// TIA Portal V19 export
FUNCTION_BLOCK "A0302_Rulliera_FB"   // FB64, LAD
// stored: MemoryReserve 100, SetENOAutomatically false
   VAR_INPUT
      AreaInterface : "AreaInterface";
      ZSI : "udt_ZoneSafetyInterface";
      DSI_Feed1 : "udt_DeviceSafetyInterface";
      DSI_Feed2 : "udt_DeviceSafetyInterface";
      Drive_Ax1 : "TAx_DriveInterface";
      Drive_Ax2 : "TAx_DriveInterface";
      DataIn : Struct
         Ax : "SpeedMachine_DataIn";
         Sens : Struct
            Coda { ExternalAccessible := 'False'; ExternalVisible := 'False'; ExternalWritable := 'False'} : Struct
               FTC_Rall : Bool;   // Sensori presenza materiale banco rallentamento ingresso
               FTC_Prox_Ing : Bool;   // Sensori presenza materiale banco limite ingresso
            END_STRUCT;
            Centro { ExternalAccessible := 'False'; ExternalVisible := 'False'; ExternalWritable := 'False'} : Struct
               FTC_Centrale : Bool;
            END_STRUCT;
         END_STRUCT;
      END_STRUCT;
      CIn { ExternalAccessible := 'False'; ExternalVisible := 'False'; ExternalWritable := 'False'} : Struct
         Manager : Struct
            Ax_1 : "SpeedMachine_CIn_Manager";
            Ax_2 : "SpeedMachine_CIn_Manager";
         END_STRUCT;
         SemiAut_Pb : Bool;
         P5 : Struct
            Sollevatori : "ValveMachine_COut";
            SpintoreLong : "ValveMachine_COut";
            Sens : Struct
               FTC_Ingombro_A0301 : Bool;   // 1614BF1 - I50.7
            END_STRUCT;
         END_STRUCT;
         Bordatrice : Struct
            StopBordatrice : Bool;   // Stop Bordatrice da controllo quota spazio rimanente su rulliera di coda
            ReadyForMove : Bool;   // Pronto al movimento
            StandbyBordatrice : Bool;
         END_STRUCT;
         Rulliera : Struct
            Centratori : "ValveMachine_COut";   // Chiusura Centratori
            Sollevamento : "ValveMachine_COut";   // Solleva centratori
            Coda : Struct
               Sens : Struct
                  FTC_Rall : Bool;   // Sensori presenza materiale banco rallentamento ingresso
                  FTC_Prox_Ing : Bool;   // Sensori presenza materiale banco limite ingresso
               END_STRUCT;
            END_STRUCT;
            Centro : Struct
               Sens : Struct
                  FTC_Centrale : Bool;   // 2010BF1 - I50.2
               END_STRUCT;
            END_STRUCT;
         END_STRUCT;
         CarroPareggCoda : Struct
            Ax : "Positioning_DOL_Machine_COut";
            Bloccaggio : "ValveMachine_COut";
            BattutaVerticale : "ValveMachine_COut";
            PareggiatoreLong : "ValveMachine_COut";
            Sens : Struct
               FTC_Ingombro_In : Bool;   // 2012BF1 - I50.0
               FTC_Ingombro_Out : Bool;   // 2012BF2 - I50.1
               PresenzaMat : Bool;   // FC presenza materiale agganciato lato paregg coda
               PosPareggLong : Struct
                  Value : LReal;
                  CheckMeasure : Bool;
                  Standstill : Bool;
               END_STRUCT;
            END_STRUCT;
         END_STRUCT;
         CarroPareggTesta : Struct
            Ax : "Positioning_DOL_Machine_COut";
            Bloccaggio : "ValveMachine_COut";
            Centraggio : "ValveMachine_COut";
            Sollevatore : "ValveMachine_COut";
            Sens : Struct
               FTC1_Rall : Bool;   // 2010BF2 - I50.3
               FTC2_Prox_Ls : Bool;   // 2010BF3 - I50.4
               PresenzaMat : Bool;   // FC presenza materiale agganciato lato paregg testa
            END_STRUCT;
         END_STRUCT;
         BTrk : Struct
            ZoneA0302Entry_Empty : Bool;
            ZoneA0302Exit_Empty : Bool;
         END_STRUCT;
      END_STRUCT;
      Config : Struct
         Ax : "SpeedMachine_Config";
      END_STRUCT;
      HWID_Ax_TEL1 : Array[1..2] of HW_SUBMODULE;
   END_VAR
   VAR_OUTPUT
      MachineInterface : "MachineInterface";
      COut : Struct
         Ax_1 : "SpeedMachine_COut";
         Ax_2 : "SpeedMachine_COut";
         Ax_VelOveride : Struct
            Enable : Bool;
            Value : Real;
         END_STRUCT;
      END_STRUCT;
   END_VAR
   VAR_IN_OUT
      Par : Struct
         Ax : "SpeedMachine_Par";
         Ax_Aut : "A0301_Mach_Speed_Par";
      END_STRUCT;
      IEC_SP : Struct
         FTC_CodaRall : Struct
            TON_PT : Time;
            TOF_PT : Time;
         END_STRUCT;
         FTC_CodaProx_Ing : Struct
            TON_PT : Time;
            TOF_PT : Time;
         END_STRUCT;
         FTC_Centro : Struct
            TON_PT : Time;
            TOF_PT : Time;
         END_STRUCT;
      END_STRUCT;
   END_VAR
   VAR
      Alarm : Struct
         Rulliera : Array[1..2] of "SpeedMachine_Alr";
      END_STRUCT;
      Warning : Struct
         Rulliera : Array[1..2] of "SpeedMachine_Wng";
         OP_REST_MissingCnd : Bool;   // Mancanza comando arresto
         OP_WORK_MissingCnd : Bool;   // Mancanza consenso lavoro
      END_STRUCT;
      HMI : Struct
         Selection : Struct   // 0=Disable / 1=Enable Pin
            Ax : Int;   // 0:Entrambe / 1:Rulliera Ax1 / 2:Rulliera Ax2
         END_STRUCT;
      END_STRUCT;
      Ax_1 : "SpeedMachine_FB";
      Ax_2 : "SpeedMachine_FB";
      ValueVelOvr { ExternalAccessible := 'False'; ExternalVisible := 'False'; ExternalWritable := 'False'} : Array[1..10] of Real;
      Sts : Struct
         OP_CanMoveFreely : Bool;
         OP_Bwd_Cnd : Bool;
         OP_Fwd_Cnd : Bool;
      END_STRUCT;
      Ctrl : Struct
         OP_Bwd_Man : Bool;
         OP_Fwd_Man : Bool;
         OP_Bwd_Aut : Bool;
         OP_Fwd_Aut : Bool;
         OP_Bwd_Run : Bool;
         OP_Fwd_Run : Bool;
      END_STRUCT;
      AUX : Struct
         OP_Bwd_PB : Bool;
         OP_Fwd_PB : Bool;
      END_STRUCT;
      TON_OP_REST_MissingCnd { S7_SetPoint := 'True'} : TON_TIME;
      TON_OP_WORK_MissingCnd { S7_SetPoint := 'True'} : TON_TIME;
      IEC_FTC_CodaRall : Struct
         TON_Delay : IEC_TIMER;
         TOF_Delay { S7_SetPoint := 'True'} : IEC_TIMER;
         FTC_On { S7_SetPoint := 'True'} : Bool;
      END_STRUCT;
      IEC_FTC_CodaProxIng : Struct
         TON_Delay : IEC_TIMER;
         TOF_Delay { S7_SetPoint := 'True'} : IEC_TIMER;
         FTC_On { S7_SetPoint := 'True'} : Bool;
      END_STRUCT;
      IEC_FTC_Centro : Struct
         TON_Delay : IEC_TIMER;
         TOF_Delay { S7_SetPoint := 'True'} : IEC_TIMER;
         FTC_On { S7_SetPoint := 'True'} : Bool;
      END_STRUCT;
   END_VAR
   VAR_TEMP
      PE : Struct
         OP_Bwd_PB : Bool;
         OP_Fwd_PB : Bool;
      END_STRUCT;
      VelOvr_Max : Real;   // Velocità max trovata
      i : Int;
      Check : Struct
         Cndz1_StartFwd : Bool;   // Check conditions to P4
         Cndz2_StartFwd : Bool;   // Check conditions to Allineatore laterale
      END_STRUCT;
   END_VAR
   VAR_TEMP   // added for the SCL form of the ladder/FBD networks
      _w1 : Bool;
      _w2 : Bool;
      _w3 : Bool;
   END_VAR
BEGIN

REGION Network 1 (SCL): == Riferimenti [Ax] - Speed Machine ==
   // ******************************************************************************************
   REGION // TRASFERIMENTO DELLE RAMPE

       // Rampe in Manuale
       IF #AreaInterface.Man AND NOT #CIn.SemiAut_Pb THEN
           #Ax_1.CIn.Manager.Vel := #Ax_2.CIn.Manager.Vel := #Par.Ax.Man.VelFwdHigh;
           #Ax_1.CIn.Manager.Acc :=  #Ax_2.CIn.Manager.Acc := #Par.Ax.Man.Acc;
           #Ax_1.CIn.Manager.Dec := #Ax_2.CIn.Manager.Dec := #Par.Ax.Man.Dec;
       END_IF;
   END_REGION

   // ******************************************************************************************
   REGION // CALCOLO DELLA VELOCITA' TRASFERITA DALL'IMPIANTO IN BASE ALLA LUNGHEZZA DEL PEZZO 

       // Inizializzo variabile di appoggio controllo overide massimo a un valore basso rispetto setpoint
       IF "Sys".AuxFirstPLCCycle THEN
           #VelOvr_Max := 100.0;
       END_IF;

       // Trasferisco le varibili su un array
       #ValueVelOvr[1] := "PPrf_MAIN".ON_WORK.A0301_A0302.Trasporto.VelOvr_PLen_UpTo_1000;
       #ValueVelOvr[2] := "PPrf_MAIN".ON_WORK.A0301_A0302.Trasporto.VelOvr_PLen_UpTo_1500;
       #ValueVelOvr[3] := "PPrf_MAIN".ON_WORK.A0301_A0302.Trasporto.VelOvr_PLen_UpTo_2000;
       #ValueVelOvr[4] := "PPrf_MAIN".ON_WORK.A0301_A0302.Trasporto.VelOvr_PLen_UpTo_2500;
       #ValueVelOvr[5] := "PPrf_MAIN".ON_WORK.A0301_A0302.Trasporto.VelOvr_PLen_UpTo_3000;
       #ValueVelOvr[6] := "PPrf_MAIN".ON_WORK.A0301_A0302.Trasporto.VelOvr_PLen_UpTo_3500;
       #ValueVelOvr[7] := "PPrf_MAIN".ON_WORK.A0301_A0302.Trasporto.VelOvr_PLen_UpTo_4000;
       #ValueVelOvr[8] := "PPrf_MAIN".ON_WORK.A0301_A0302.Trasporto.VelOvr_PLen_UpTo_4500;
       #ValueVelOvr[9] := "PPrf_MAIN".ON_WORK.A0301_A0302.Trasporto.VelOvr_PLen_UpTo_5000;
       #ValueVelOvr[10] := "PPrf_MAIN".ON_WORK.A0301_A0302.Trasporto.VelOvr_PLen_UpTo_5500;


       // Ciclo per verificare la variabile maggiore per prenderla in lavoro
       FOR #i := 1 TO 10 DO
           IF #ValueVelOvr[#i] >= #VelOvr_Max THEN
               #VelOvr_Max := #ValueVelOvr[#i];
           END_IF;
       END_FOR;
   END_REGION ;

   IF #VelOvr_Max = 0.0 THEN
       #VelOvr_Max := 100.0;
   END_IF;

   // ******************************************************************************************
   REGION // CALCOLO DELLA VELOCITA' E TRASFERIMENTO IN BASE ALLO STATO IMPIANTO

       #Ax_1.CIn.VelocityOverride.Enable := TRUE;
       #Ax_2.CIn.VelocityOverride.Enable := TRUE;

       IF #Ax_1.CIn.Manager.Control_ON THEN
           // CALCOLO VELOCITA' IN BASE ALL'OVERIDE
           #Ax_1.CIn.VelocityOverride.Value :=  #VelOvr_Max;
       ELSE
           #Ax_1.CIn.VelocityOverride.Value := 100.0;
           END_IF;

           IF #Ax_2.CIn.Manager.Control_ON THEN
               #Ax_2.CIn.VelocityOverride.Value := #VelOvr_Max;
           ELSE
               #Ax_2.CIn.VelocityOverride.Value := 100.0;
           END_IF;
       END_REGION ;
END_REGION

REGION Network 3: DataIn - FTC CodaRall
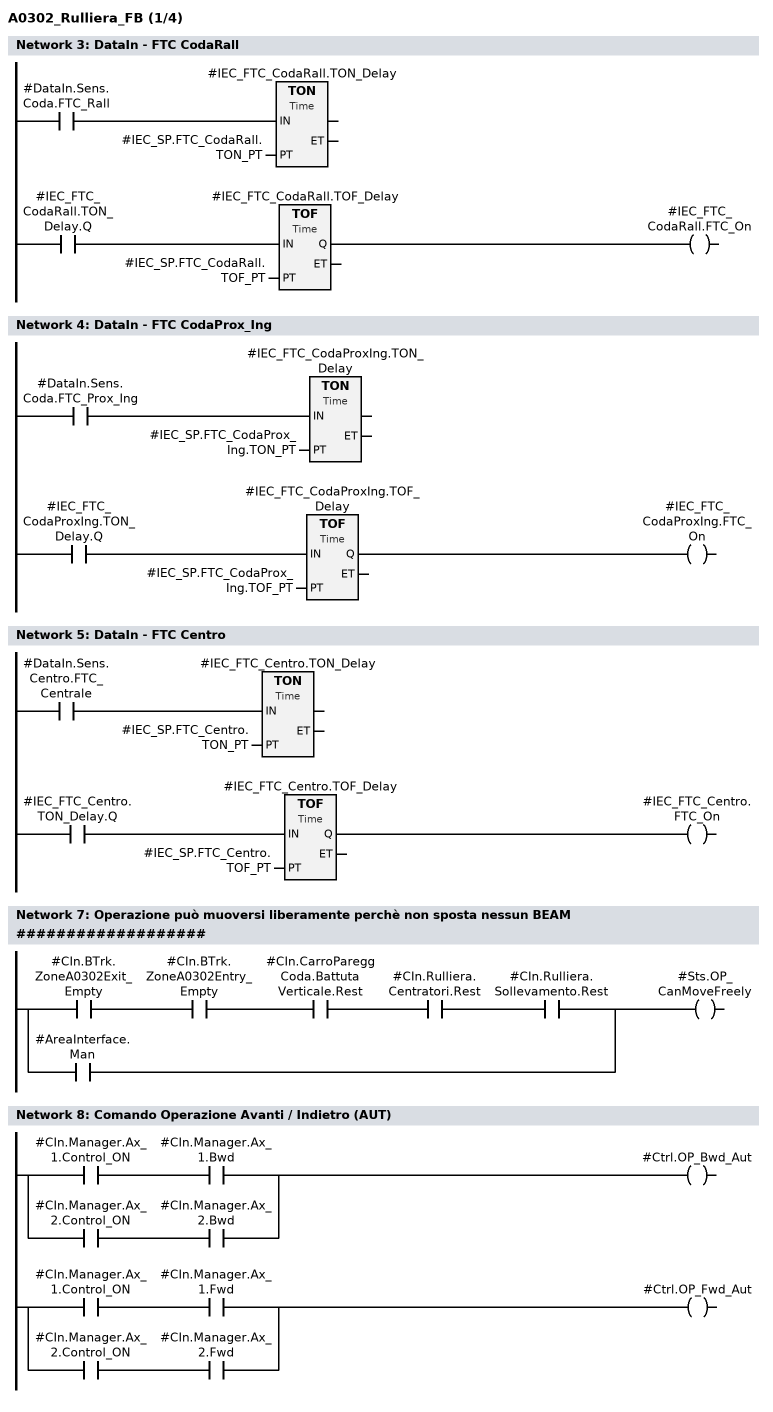
   RUNG wire#powerrail
      Contact( #DataIn.Sens.Coda.FTC_Rall )
      { S7_Templates := "time_type := Time" } #IEC_FTC_CodaRall.TON_Delay.TON(pt := #IEC_SP.FTC_CodaRall.TON_PT, et =>)
   END_RUNG
   RUNG wire#powerrail
      Contact( #IEC_FTC_CodaRall.TON_Delay.Q )
      { S7_Templates := "time_type := Time" } #IEC_FTC_CodaRall.TOF_Delay.TOF(pt := #IEC_SP.FTC_CodaRall.TOF_PT, et =>)
      Coil( #IEC_FTC_CodaRall.FTC_On )
   END_RUNG
   // the same network as SCL:
   #IEC_FTC_CodaRall.TON_Delay.TON(IN := #DataIn.Sens.Coda.FTC_Rall, PT := #IEC_SP.FTC_CodaRall.TON_PT);
   #IEC_FTC_CodaRall.TOF_Delay.TOF(IN := #IEC_FTC_CodaRall.TON_Delay.Q, PT := #IEC_SP.FTC_CodaRall.TOF_PT);
   #IEC_FTC_CodaRall.FTC_On := #IEC_FTC_CodaRall.TOF_Delay.Q;
END_REGION

REGION Network 4: DataIn - FTC CodaProx_Ing
   RUNG wire#powerrail
      Contact( #DataIn.Sens.Coda.FTC_Prox_Ing )
      { S7_Templates := "time_type := Time" } #IEC_FTC_CodaProxIng.TON_Delay.TON(pt := #IEC_SP.FTC_CodaProx_Ing.TON_PT, et =>)
   END_RUNG
   RUNG wire#powerrail
      Contact( #IEC_FTC_CodaProxIng.TON_Delay.Q )
      { S7_Templates := "time_type := Time" } #IEC_FTC_CodaProxIng.TOF_Delay.TOF(pt := #IEC_SP.FTC_CodaProx_Ing.TOF_PT, et =>)
      Coil( #IEC_FTC_CodaProxIng.FTC_On )
   END_RUNG
   // the same network as SCL:
   #IEC_FTC_CodaProxIng.TON_Delay.TON(IN := #DataIn.Sens.Coda.FTC_Prox_Ing,
                           PT := #IEC_SP.FTC_CodaProx_Ing.TON_PT);
   #IEC_FTC_CodaProxIng.TOF_Delay.TOF(IN := #IEC_FTC_CodaProxIng.TON_Delay.Q,
                           PT := #IEC_SP.FTC_CodaProx_Ing.TOF_PT);
   #IEC_FTC_CodaProxIng.FTC_On := #IEC_FTC_CodaProxIng.TOF_Delay.Q;
END_REGION

REGION Network 5: DataIn - FTC Centro
   RUNG wire#powerrail
      Contact( #DataIn.Sens.Centro.FTC_Centrale )
      { S7_Templates := "time_type := Time" } #IEC_FTC_Centro.TON_Delay.TON(pt := #IEC_SP.FTC_Centro.TON_PT, et =>)
   END_RUNG
   RUNG wire#powerrail
      Contact( #IEC_FTC_Centro.TON_Delay.Q )
      { S7_Templates := "time_type := Time" } #IEC_FTC_Centro.TOF_Delay.TOF(pt := #IEC_SP.FTC_Centro.TOF_PT, et =>)
      Coil( #IEC_FTC_Centro.FTC_On )
   END_RUNG
   // the same network as SCL:
   #IEC_FTC_Centro.TON_Delay.TON(IN := #DataIn.Sens.Centro.FTC_Centrale, PT := #IEC_SP.FTC_Centro.TON_PT);
   #IEC_FTC_Centro.TOF_Delay.TOF(IN := #IEC_FTC_Centro.TON_Delay.Q, PT := #IEC_SP.FTC_Centro.TOF_PT);
   #IEC_FTC_Centro.FTC_On := #IEC_FTC_Centro.TOF_Delay.Q;
END_REGION

REGION Network 7: Operazione può muoversi liberamente perchè non sposta nessun BEAM ###################
   RUNG wire#powerrail
      Contact( #CIn.BTrk.ZoneA0302Exit_Empty )
      Contact( #CIn.BTrk.ZoneA0302Entry_Empty )
      Contact( #CIn.CarroPareggCoda.BattutaVerticale.Rest )
      Contact( #CIn.Rulliera.Centratori.Rest )
      Contact( #CIn.Rulliera.Sollevamento.Rest )
      wire#w1
      Coil( #Sts.OP_CanMoveFreely )
   END_RUNG
   RUNG wire#powerrail
      Contact( #AreaInterface.Man )
   END_RUNG wire#w1
   // the same network as SCL:
   #Sts.OP_CanMoveFreely := (#CIn.BTrk.ZoneA0302Exit_Empty AND #CIn.BTrk.ZoneA0302Entry_Empty AND #CIn.CarroPareggCoda.BattutaVerticale.Rest AND #CIn.Rulliera.Centratori.Rest AND #CIn.Rulliera.Sollevamento.Rest) OR #AreaInterface.Man;
END_REGION

REGION Network 8: Comando Operazione Avanti / Indietro (AUT)
   RUNG wire#powerrail
      Contact( #CIn.Manager.Ax_1.Control_ON )
      Contact( #CIn.Manager.Ax_1.Bwd )
      wire#w1
      Coil( #Ctrl.OP_Bwd_Aut )
   END_RUNG
   RUNG wire#powerrail
      Contact( #CIn.Manager.Ax_2.Control_ON )
      Contact( #CIn.Manager.Ax_2.Bwd )
   END_RUNG wire#w1
   RUNG wire#powerrail
      Contact( #CIn.Manager.Ax_1.Control_ON )
      Contact( #CIn.Manager.Ax_1.Fwd )
      wire#w2
      Coil( #Ctrl.OP_Fwd_Aut )
   END_RUNG
   RUNG wire#powerrail
      Contact( #CIn.Manager.Ax_2.Control_ON )
      Contact( #CIn.Manager.Ax_2.Fwd )
   END_RUNG wire#w2
   // the same network as SCL:
   #Ctrl.OP_Bwd_Aut := (#CIn.Manager.Ax_1.Control_ON AND #CIn.Manager.Ax_1.Bwd) OR (#CIn.Manager.Ax_2.Control_ON AND #CIn.Manager.Ax_2.Bwd);
   #Ctrl.OP_Fwd_Aut := (#CIn.Manager.Ax_1.Control_ON AND #CIn.Manager.Ax_1.Fwd) OR (#CIn.Manager.Ax_2.Control_ON AND #CIn.Manager.Ax_2.Fwd);
END_REGION

REGION Network 9: Comando Operazione Lavoro / Riposo (MAN)
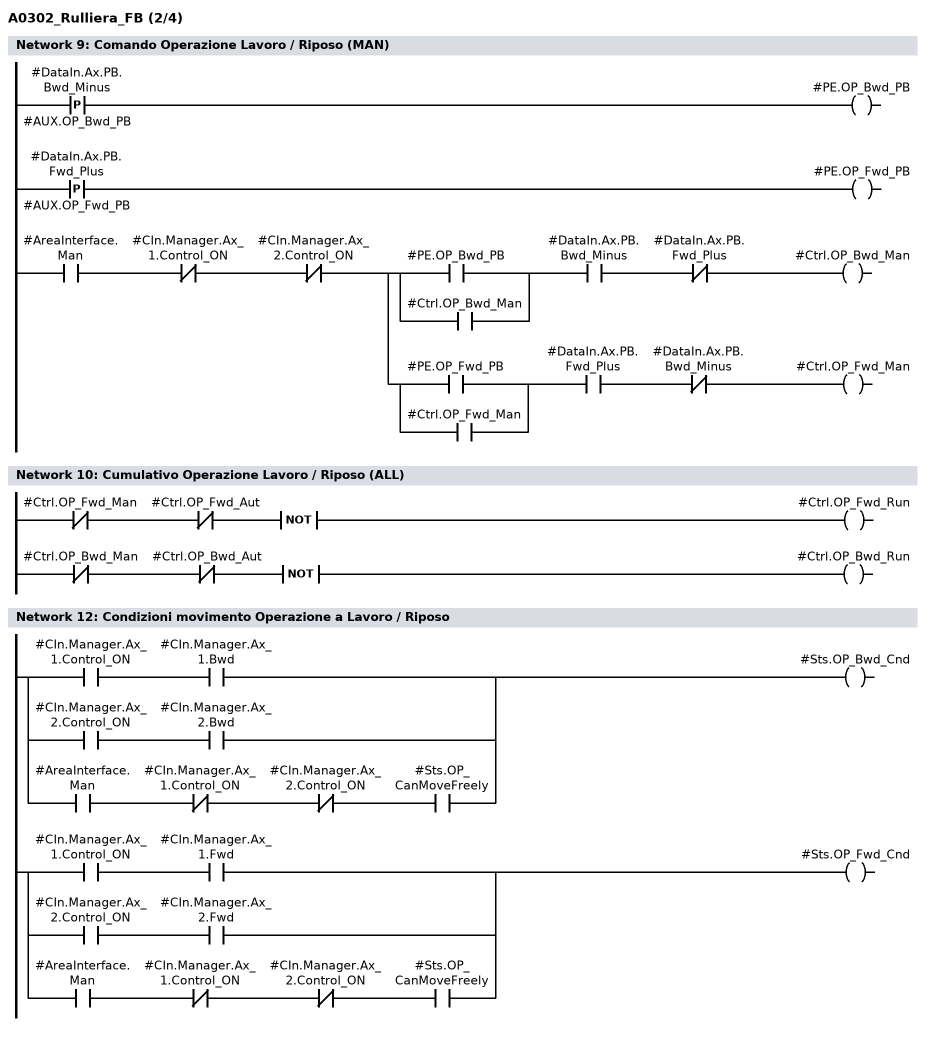
   RUNG wire#powerrail
      P_Contact(operand := #DataIn.Ax.PB.Bwd_Minus, bit := #AUX.OP_Bwd_PB)
      Coil( #PE.OP_Bwd_PB )
   END_RUNG
   RUNG wire#powerrail
      P_Contact(operand := #DataIn.Ax.PB.Fwd_Plus, bit := #AUX.OP_Fwd_PB)
      Coil( #PE.OP_Fwd_PB )
   END_RUNG
   RUNG wire#powerrail
      Contact( #AreaInterface.Man )
      I_Contact( #CIn.Manager.Ax_1.Control_ON )
      I_Contact( #CIn.Manager.Ax_2.Control_ON )
      wire#w1
      Contact( #PE.OP_Bwd_PB )
      wire#w2
      Contact( #DataIn.Ax.PB.Bwd_Minus )
      I_Contact( #DataIn.Ax.PB.Fwd_Plus )
      Coil( #Ctrl.OP_Bwd_Man )
   END_RUNG
   RUNG wire#w1
      Contact( #Ctrl.OP_Bwd_Man )
   END_RUNG wire#w2
   RUNG wire#w1
      Contact( #PE.OP_Fwd_PB )
      wire#w3
      Contact( #DataIn.Ax.PB.Fwd_Plus )
      I_Contact( #DataIn.Ax.PB.Bwd_Minus )
      Coil( #Ctrl.OP_Fwd_Man )
   END_RUNG
   RUNG wire#w1
      Contact( #Ctrl.OP_Fwd_Man )
   END_RUNG wire#w3
   // the same network as SCL:
   #_w1 := #DataIn.Ax.PB.Bwd_Minus AND NOT #AUX.OP_Bwd_PB;   // rising edge of #DataIn.Ax.PB.Bwd_Minus
   #AUX.OP_Bwd_PB := #DataIn.Ax.PB.Bwd_Minus;
   #PE.OP_Bwd_PB := #_w1;
   #_w2 := #DataIn.Ax.PB.Fwd_Plus AND NOT #AUX.OP_Fwd_PB;   // rising edge of #DataIn.Ax.PB.Fwd_Plus
   #AUX.OP_Fwd_PB := #DataIn.Ax.PB.Fwd_Plus;
   #PE.OP_Fwd_PB := #_w2;
   #_w3 := #AreaInterface.Man AND NOT #CIn.Manager.Ax_1.Control_ON AND NOT #CIn.Manager.Ax_2.Control_ON;
   #Ctrl.OP_Bwd_Man := #_w3 AND (#PE.OP_Bwd_PB OR #Ctrl.OP_Bwd_Man) AND #DataIn.Ax.PB.Bwd_Minus AND NOT #DataIn.Ax.PB.Fwd_Plus;
   #Ctrl.OP_Fwd_Man := #_w3 AND (#PE.OP_Fwd_PB OR #Ctrl.OP_Fwd_Man) AND #DataIn.Ax.PB.Fwd_Plus AND NOT #DataIn.Ax.PB.Bwd_Minus;
END_REGION

REGION Network 10: Cumulativo Operazione Lavoro / Riposo (ALL)
   RUNG wire#powerrail
      I_Contact( #Ctrl.OP_Fwd_Man )
      I_Contact( #Ctrl.OP_Fwd_Aut )
      Not()
      Coil( #Ctrl.OP_Fwd_Run )
   END_RUNG
   RUNG wire#powerrail
      I_Contact( #Ctrl.OP_Bwd_Man )
      I_Contact( #Ctrl.OP_Bwd_Aut )
      Not()
      Coil( #Ctrl.OP_Bwd_Run )
   END_RUNG
   // the same network as SCL:
   #Ctrl.OP_Fwd_Run := NOT (NOT #Ctrl.OP_Fwd_Man AND NOT #Ctrl.OP_Fwd_Aut);
   #Ctrl.OP_Bwd_Run := NOT (NOT #Ctrl.OP_Bwd_Man AND NOT #Ctrl.OP_Bwd_Aut);
END_REGION

REGION Network 11: <+>
END_REGION

REGION Network 12: Condizioni movimento Operazione a Lavoro / Riposo
   RUNG wire#powerrail
      Contact( #CIn.Manager.Ax_1.Control_ON )
      Contact( #CIn.Manager.Ax_1.Bwd )
      wire#w1
      Coil( #Sts.OP_Bwd_Cnd )
   END_RUNG
   RUNG wire#powerrail
      Contact( #CIn.Manager.Ax_2.Control_ON )
      Contact( #CIn.Manager.Ax_2.Bwd )
   END_RUNG wire#w1
   RUNG wire#powerrail
      Contact( #AreaInterface.Man )
      I_Contact( #CIn.Manager.Ax_1.Control_ON )
      I_Contact( #CIn.Manager.Ax_2.Control_ON )
      Contact( #Sts.OP_CanMoveFreely )
   END_RUNG wire#w1
   RUNG wire#powerrail
      Contact( #CIn.Manager.Ax_1.Control_ON )
      Contact( #CIn.Manager.Ax_1.Fwd )
      wire#w2
      Coil( #Sts.OP_Fwd_Cnd )
   END_RUNG
   RUNG wire#powerrail
      Contact( #CIn.Manager.Ax_2.Control_ON )
      Contact( #CIn.Manager.Ax_2.Fwd )
   END_RUNG wire#w2
   RUNG wire#powerrail
      Contact( #AreaInterface.Man )
      I_Contact( #CIn.Manager.Ax_1.Control_ON )
      I_Contact( #CIn.Manager.Ax_2.Control_ON )
      Contact( #Sts.OP_CanMoveFreely )
   END_RUNG wire#w2
   // the same network as SCL:
   #Sts.OP_Bwd_Cnd := (#CIn.Manager.Ax_1.Control_ON AND #CIn.Manager.Ax_1.Bwd) OR (#CIn.Manager.Ax_2.Control_ON AND #CIn.Manager.Ax_2.Bwd) OR (#AreaInterface.Man AND NOT #CIn.Manager.Ax_1.Control_ON AND NOT #CIn.Manager.Ax_2.Control_ON AND #Sts.OP_CanMoveFreely);
   #Sts.OP_Fwd_Cnd := (#CIn.Manager.Ax_1.Control_ON AND #CIn.Manager.Ax_1.Fwd) OR (#CIn.Manager.Ax_2.Control_ON AND #CIn.Manager.Ax_2.Fwd) OR (#AreaInterface.Man AND NOT #CIn.Manager.Ax_1.Control_ON AND NOT #CIn.Manager.Ax_2.Control_ON AND #Sts.OP_CanMoveFreely);
END_REGION

REGION Network 13 (SCL): [Ax_1 + Ax_2] - CIn Manger
   // TRASFERIMENTO CIn MANAGER ALLA MACCHINA
   #Ax_1.CIn.Manager := #CIn.Manager.Ax_1;
   #Ax_2.CIn.Manager := #CIn.Manager.Ax_2;
END_REGION

REGION Network 14 (SCL): [Ax_1 + Ax_2] - Cin Manager Comando arresto / lavoro
   //
   #Ax_1.CIn.Manager.Bwd := #Ax_2.CIn.Manager.Bwd := FALSE;
   //************************************
   #Ax_1.CIn.Manager.Fwd := #Ax_2.CIn.Manager.Fwd := FALSE;
   //
   // CIn Manager  Control ON se ho un richiesta di comando attiva
   #Ax_1.CIn.Manager.Control_ON := #Ax_2.CIn.Manager.Control_ON := #Ctrl.OP_Fwd_Run OR #Ctrl.OP_Bwd_Run;

   // CIn Manager Brw se ho un richiesta di comando indietro attiva
   #Ax_1.CIn.Manager.Bwd := #Ax_2.CIn.Manager.Bwd := #Ctrl.OP_Bwd_Run AND #Sts.OP_Bwd_Cnd;

   // CIn Manager Frw se ho un richiesta di comando avanti attiva
   // Se la battuta di coda è alta attivo tutte e 2 le rulliere
   IF #Ctrl.OP_Fwd_Run AND #Sts.OP_Fwd_Cnd AND #CIn.CarroPareggCoda.BattutaVerticale.Rest THEN
       #Ax_1.CIn.Manager.Fwd := #Ax_2.CIn.Manager.Fwd := TRUE;


       // Se la battuta di coda è bassa attivo la rulliera 1 e la 2 rimane ferma
   ELSIF (#Ctrl.OP_Fwd_Run AND #Sts.OP_Fwd_Cnd) AND #CIn.CarroPareggCoda.BattutaVerticale.Work THEN
       #Ax_1.CIn.Manager.Fwd := TRUE;
       #Ax_2.CIn.Manager.Fwd := FALSE;
   END_IF;
END_REGION

REGION Network 15 (SCL): [Ax_1 + 2] - CIn Abilitazioni Stop Manager
   // CIn Manager Stop per richiesta apertura safety
   // 
   #Ax_1.CIn.Manager.EnableStopDoorOpeningReq := #CIn.Manager.Ax_1.EnableStopDoorOpeningReq;
   #Ax_2.CIn.Manager.EnableStopDoorOpeningReq := #CIn.Manager.Ax_2.EnableStopDoorOpeningReq;

   // CIn Manager Stop in fase delle macchine precedenti
   // 
   #Ax_1.CIn.Manager.EnableStopInPhase := #CIn.Manager.Ax_1.EnableStopInPhase;
   #Ax_2.CIn.Manager.EnableStopInPhase := #CIn.Manager.Ax_2.EnableStopInPhase;

   // CIn Manager Stop programmato configurabile a piacere
   // 
   #Ax_1.CIn.Manager.EnableStopProgrammed := #CIn.Manager.Ax_1.EnableStopProgrammed;
   #Ax_2.CIn.Manager.EnableStopProgrammed := #CIn.Manager.Ax_2.EnableStopProgrammed;
END_REGION

REGION Network 16: <+>
END_REGION

REGION Network 17: Warning manacanza condizioni esecuzione Operazione RIPOSO / LAVORO
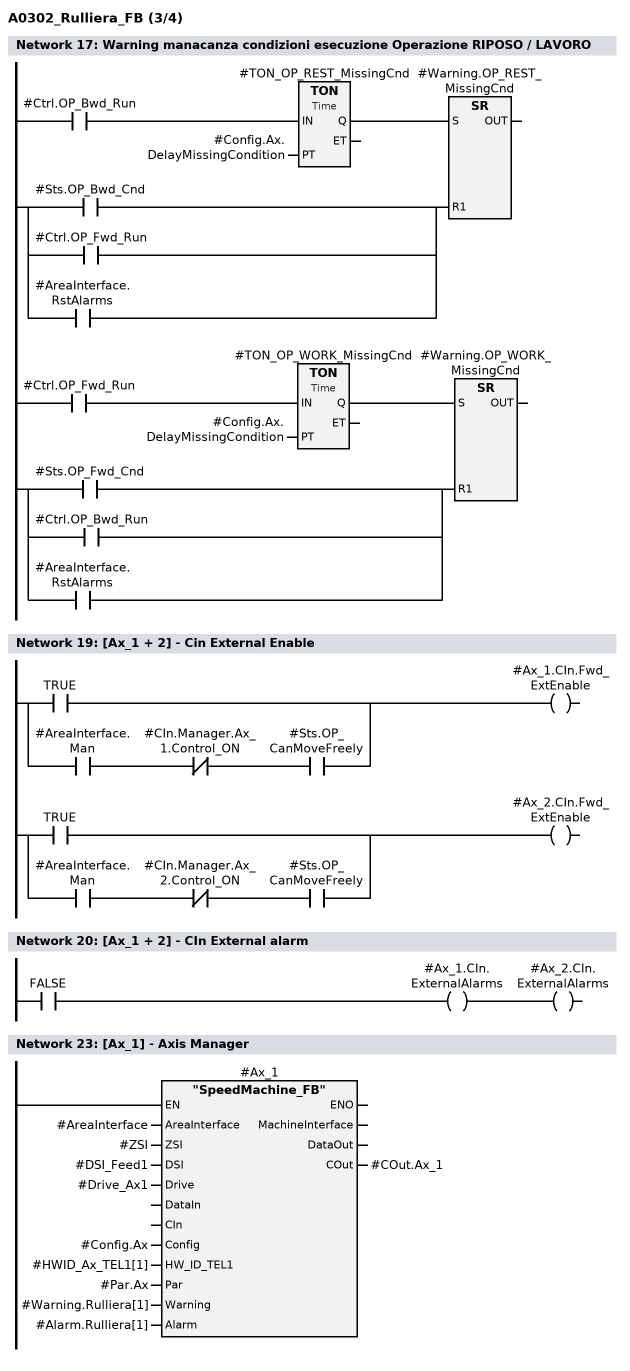
   RUNG wire#powerrail
      Contact( #Ctrl.OP_Bwd_Run )
      { S7_Templates := "time_type := Time" } #TON_OP_REST_MissingCnd.TON(pt := #Config.Ax.DelayMissingCondition, et =>)
      S_SR(operand := #Warning.OP_REST_MissingCnd, r1 := wire#w1)
   END_RUNG
   RUNG wire#powerrail
      Contact( #Sts.OP_Bwd_Cnd )
   END_RUNG wire#w1
   RUNG wire#powerrail
      Contact( #Ctrl.OP_Fwd_Run )
   END_RUNG wire#w1
   RUNG wire#powerrail
      Contact( #AreaInterface.RstAlarms )
   END_RUNG wire#w1
   RUNG wire#powerrail
      Contact( #Ctrl.OP_Fwd_Run )
      { S7_Templates := "time_type := Time" } #TON_OP_WORK_MissingCnd.TON(pt := #Config.Ax.DelayMissingCondition, et =>)
      S_SR(operand := #Warning.OP_WORK_MissingCnd, r1 := wire#w2)
   END_RUNG
   RUNG wire#powerrail
      Contact( #Sts.OP_Fwd_Cnd )
   END_RUNG wire#w2
   RUNG wire#powerrail
      Contact( #Ctrl.OP_Bwd_Run )
   END_RUNG wire#w2
   RUNG wire#powerrail
      Contact( #AreaInterface.RstAlarms )
   END_RUNG wire#w2
   // the same network as SCL:
   #TON_OP_REST_MissingCnd(IN := #Ctrl.OP_Bwd_Run, PT := #Config.Ax.DelayMissingCondition);   // TON
   IF #TON_OP_REST_MissingCnd.Q THEN
       #Warning.OP_REST_MissingCnd := TRUE;   // SR flip-flop
   END_IF;
   IF #Sts.OP_Bwd_Cnd OR #Ctrl.OP_Fwd_Run OR #AreaInterface.RstAlarms THEN
       #Warning.OP_REST_MissingCnd := FALSE;
   END_IF;
   #TON_OP_WORK_MissingCnd(IN := #Ctrl.OP_Fwd_Run, PT := #Config.Ax.DelayMissingCondition);   // TON
   IF #TON_OP_WORK_MissingCnd.Q THEN
       #Warning.OP_WORK_MissingCnd := TRUE;   // SR flip-flop
   END_IF;
   IF #Sts.OP_Fwd_Cnd OR #Ctrl.OP_Bwd_Run OR #AreaInterface.RstAlarms THEN
       #Warning.OP_WORK_MissingCnd := FALSE;
   END_IF;
END_REGION

REGION Network 18: <+>
END_REGION

REGION Network 19: [Ax_1 + 2] - Cin External Enable
   RUNG wire#powerrail
      Contact( TRUE )
      wire#w1
      Coil( #Ax_1.CIn.Fwd_ExtEnable )
   END_RUNG
   RUNG wire#powerrail
      Contact( #AreaInterface.Man )
      I_Contact( #CIn.Manager.Ax_1.Control_ON )
      Contact( #Sts.OP_CanMoveFreely )
   END_RUNG wire#w1
   RUNG wire#powerrail
      Contact( TRUE )
      wire#w2
      Coil( #Ax_2.CIn.Fwd_ExtEnable )
   END_RUNG
   RUNG wire#powerrail
      Contact( #AreaInterface.Man )
      I_Contact( #CIn.Manager.Ax_2.Control_ON )
      Contact( #Sts.OP_CanMoveFreely )
   END_RUNG wire#w2
   // the same network as SCL:
   #Ax_1.CIn.Fwd_ExtEnable := TRUE OR (#AreaInterface.Man AND NOT #CIn.Manager.Ax_1.Control_ON AND #Sts.OP_CanMoveFreely);
   #Ax_2.CIn.Fwd_ExtEnable := TRUE OR (#AreaInterface.Man AND NOT #CIn.Manager.Ax_2.Control_ON AND #Sts.OP_CanMoveFreely);
END_REGION

REGION Network 20: [Ax_1 + 2] - CIn External alarm
   RUNG wire#powerrail
      Contact( FALSE )
      Coil( #Ax_1.CIn.ExternalAlarms )
      Coil( #Ax_2.CIn.ExternalAlarms )
   END_RUNG
   // the same network as SCL:
   #Ax_1.CIn.ExternalAlarms := FALSE;
   #Ax_2.CIn.ExternalAlarms := FALSE;
END_REGION

REGION Network 21: <+>
END_REGION

REGION Network 22: <<< RULLIERA 1 >>>
END_REGION

REGION Network 23: [Ax_1] - Axis Manager
   RUNG wire#powerrail
      #Ax_1(AreaInterface := #AreaInterface, ZSI := #ZSI, DSI := #DSI_Feed1, Drive := #Drive_Ax1, DataIn :=, CIn :=, Config := #Config.Ax, HW_ID_TEL1 := #HWID_Ax_TEL1[1], Par := #Par.Ax, Warning := #Warning.Rulliera[1], Alarm := #Alarm.Rulliera[1], MachineInterface =>, DataOut =>, COut => #COut.Ax_1)
   END_RUNG
   // the same network as SCL:
   #Ax_1(AreaInterface := #AreaInterface,   // "SpeedMachine_FB"
         ZSI := #ZSI,
         DSI := #DSI_Feed1,
         Drive := #Drive_Ax1,
         Config := #Config.Ax,
         HW_ID_TEL1 := #HWID_Ax_TEL1[1],
         Par := #Par.Ax,
         Warning := #Warning.Rulliera[1],
         Alarm := #Alarm.Rulliera[1],
         COut => #COut.Ax_1);
END_REGION

REGION Network 24: <<< RULLIERA 2 >>>
END_REGION

REGION Network 25: [Ax_2] - Axis Manager
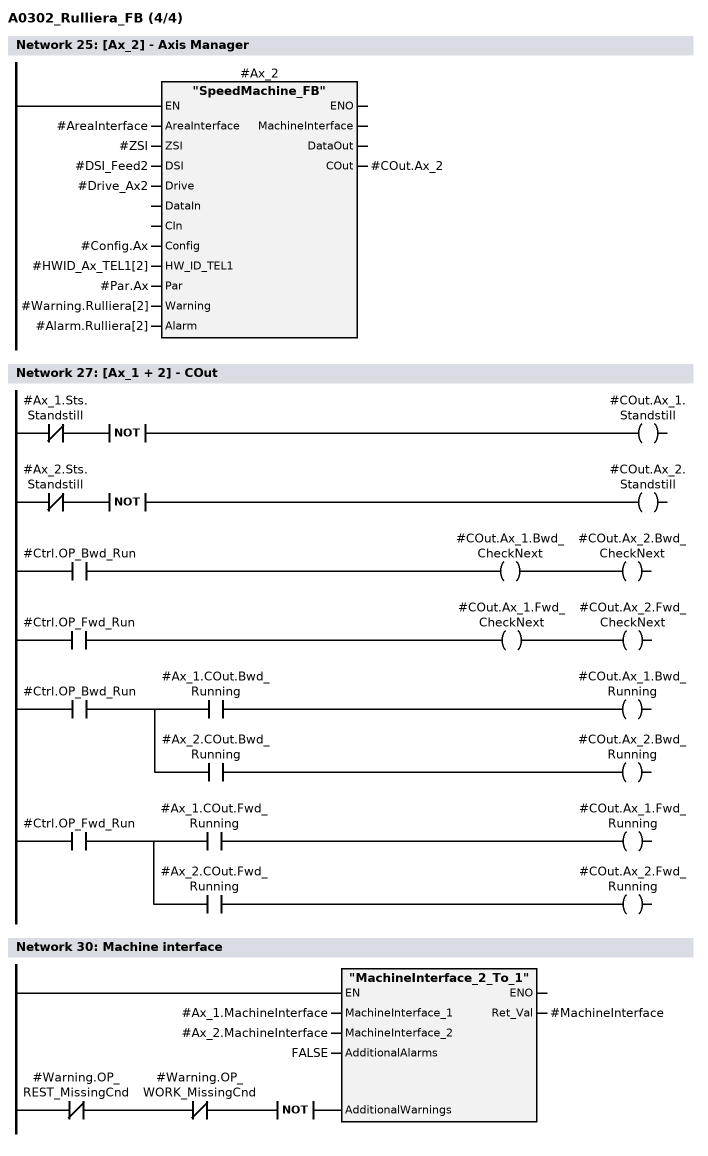
   RUNG wire#powerrail
      #Ax_2(AreaInterface := #AreaInterface, ZSI := #ZSI, DSI := #DSI_Feed2, Drive := #Drive_Ax2, DataIn :=, CIn :=, Config := #Config.Ax, HW_ID_TEL1 := #HWID_Ax_TEL1[2], Par := #Par.Ax, Warning := #Warning.Rulliera[2], Alarm := #Alarm.Rulliera[2], MachineInterface =>, DataOut =>, COut => #COut.Ax_2)
   END_RUNG
   // the same network as SCL:
   #Ax_2(AreaInterface := #AreaInterface,   // "SpeedMachine_FB"
         ZSI := #ZSI,
         DSI := #DSI_Feed2,
         Drive := #Drive_Ax2,
         Config := #Config.Ax,
         HW_ID_TEL1 := #HWID_Ax_TEL1[2],
         Par := #Par.Ax,
         Warning := #Warning.Rulliera[2],
         Alarm := #Alarm.Rulliera[2],
         COut => #COut.Ax_2);
END_REGION

REGION Network 27: [Ax_1 + 2] - COut
   RUNG wire#powerrail
      I_Contact( #Ax_1.Sts.Standstill )
      Not()
      Coil( #COut.Ax_1.Standstill )
   END_RUNG
   RUNG wire#powerrail
      I_Contact( #Ax_2.Sts.Standstill )
      Not()
      Coil( #COut.Ax_2.Standstill )
   END_RUNG
   RUNG wire#powerrail
      Contact( #Ctrl.OP_Bwd_Run )
      Coil( #COut.Ax_1.Bwd_CheckNext )
      Coil( #COut.Ax_2.Bwd_CheckNext )
   END_RUNG
   RUNG wire#powerrail
      Contact( #Ctrl.OP_Fwd_Run )
      Coil( #COut.Ax_1.Fwd_CheckNext )
      Coil( #COut.Ax_2.Fwd_CheckNext )
   END_RUNG
   RUNG wire#powerrail
      Contact( #Ctrl.OP_Bwd_Run )
      wire#w1
      Contact( #Ax_1.COut.Bwd_Running )
      Coil( #COut.Ax_1.Bwd_Running )
   END_RUNG
   RUNG wire#w1
      Contact( #Ax_2.COut.Bwd_Running )
      Coil( #COut.Ax_2.Bwd_Running )
   END_RUNG
   RUNG wire#powerrail
      Contact( #Ctrl.OP_Fwd_Run )
      wire#w2
      Contact( #Ax_1.COut.Fwd_Running )
      Coil( #COut.Ax_1.Fwd_Running )
   END_RUNG
   RUNG wire#w2
      Contact( #Ax_2.COut.Fwd_Running )
      Coil( #COut.Ax_2.Fwd_Running )
   END_RUNG
   // the same network as SCL:
   #COut.Ax_1.Standstill := NOT (NOT #Ax_1.Sts.Standstill);
   #COut.Ax_2.Standstill := NOT (NOT #Ax_2.Sts.Standstill);
   #COut.Ax_1.Bwd_CheckNext := #Ctrl.OP_Bwd_Run;
   #COut.Ax_2.Bwd_CheckNext := #Ctrl.OP_Bwd_Run;
   #COut.Ax_1.Fwd_CheckNext := #Ctrl.OP_Fwd_Run;
   #COut.Ax_2.Fwd_CheckNext := #Ctrl.OP_Fwd_Run;
   #COut.Ax_1.Bwd_Running := #Ctrl.OP_Bwd_Run AND #Ax_1.COut.Bwd_Running;
   #COut.Ax_2.Bwd_Running := #Ctrl.OP_Bwd_Run AND #Ax_2.COut.Bwd_Running;
   #COut.Ax_1.Fwd_Running := #Ctrl.OP_Fwd_Run AND #Ax_1.COut.Fwd_Running;
   #COut.Ax_2.Fwd_Running := #Ctrl.OP_Fwd_Run AND #Ax_2.COut.Fwd_Running;
END_REGION

REGION Network 29: <<< MACHINE STATUS >>>
END_REGION

REGION Network 30: Machine interface
   RUNG wire#powerrail
      "MachineInterface_2_To_1"(AdditionalWarnings := wire#w1, MachineInterface_1 := #Ax_1.MachineInterface, MachineInterface_2 := #Ax_2.MachineInterface, AdditionalAlarms := FALSE, Ret_Val => #MachineInterface)
   END_RUNG
   RUNG wire#powerrail
      I_Contact( #Warning.OP_REST_MissingCnd )
      I_Contact( #Warning.OP_WORK_MissingCnd )
      Not()
   END_RUNG wire#w1
   // the same network as SCL:
   #MachineInterface := "MachineInterface_2_To_1"(MachineInterface_1 := #Ax_1.MachineInterface,
                           MachineInterface_2 := #Ax_2.MachineInterface,
                           AdditionalAlarms := FALSE,
                           AdditionalWarnings := NOT (NOT #Warning.OP_REST_MissingCnd AND NOT #Warning.OP_WORK_MissingCnd));
END_REGION
END_FUNCTION_BLOCK
